INTERFACE ICompositeDevice EXTENDS IParentAutomationComponent, IChildAutomationComponent, IInputLeafAutomationComponent, IOutputLeafAutomationComponent

END_INTERFACE

(* stored: Version 1.1.0.1
   Itf ICompositeDevice: Id {be5e3b3f-f46a-4c0b-a57f-a0e8cfdaef93} *)
